(* IEC 61131-3 sources: ia2/library/process-control/pous (part 2) *)

(* ---- fb_pid_3step.st ---- *)
(*
  FB_PID_3STEP — step (3-step) PID: open/close pulse control of a motorized actuator,
  supporting both no-position-feedback (travel-time integral estimate) and
  with-feedback wiring.

  ~ Standard step PID / 3-step output controller (step controller / 3-step PID, driving
  integrating-type actuators such as motorized control valves and motorized dampers),
  found in every major DCS/PLC standard library.

  Purpose: closed-loop control of a motorized actuator (motorized valve / motorized
  damper, which is itself an integrating element: energized it runs open/close, de-energized
  it stops in place). Without a position transmitter, estimate position by integrating
  travel time (pos_fb < 0); with a 4-20 mA position feedback, use it directly.

  Behavior:
    1) Position estimate pos_est: pos_fb >= 0 takes the feedback directly (clamped
       0..100); otherwise integrate from the previous scan's output and the travel time:
       an open pulse adds +100*dt_s/motor_time_s, a close pulse decrements likewise
       (clamped 0..100).
    2) An internal positional PID (reverse-acting e = sp - pv, D on PV with automatic
       3*dt_s PT1 filtering) computes the target position target 0..100; integral
       back-calculation anti-windup; in manual, target tracks pos_est so the return to
       auto is bumpless. For direct-acting scenarios, invert pv/sp externally.
    3) Three-step output: position deviation = target - pos_est;
       > deadband_pct emits an open pulse, < -deadband_pct emits a close pulse, within
       the deadband stop. In auto, once a pulse is emitted it is held at least
       min_pulse_s (to avoid short pulses hammering the contactor); manual jogs
       man_open/man_close pass through (no minimum pulse width, mutually interlocked
       when both are commanded), constrained only by the travel limits. A reversal must
       pass through one scan fully stopped (stop before reversing). At a travel boundary
       (pos_est reaching 0 or 100), stop that direction's pulse immediately.
    Tuning tip: deadband_pct should be larger than the travel corresponding to the
    minimum pulse width (min_pulse_s / motor_time_s * 100%), otherwise it will still
    overshoot and oscillate within the deadband.

  Inputs:
    pv           REAL  process value
    sp           REAL  setpoint
    kp           REAL  proportional gain
    ti_s         REAL  integral time s (0 = no integral)
    td_s         REAL  derivative time s (0 = derivative off)
    dt_s         REAL  sample period s (<= 0 holds this scan, no action)
    motor_time_s REAL  actuator full-travel time s (0->100%; used for estimation and limits)
    min_pulse_s  REAL  minimum pulse width in auto s
    deadband_pct REAL  position deadband % (no action within the deviation deadband)
    auto         BOOL  TRUE auto / FALSE manual jog
    man_open     BOOL  manual open jog (interlocked, no action when commanded with man_close)
    man_close    BOOL  manual close jog
    pos_fb       REAL  position feedback 0..100 % (< 0 = no feedback, use travel estimate)
  Outputs:
    q_open  BOOL  open-direction pulse output
    q_close BOOL  close-direction pulse output
    pos_est REAL  position estimate/feedback 0..100 %
*)
FUNCTION_BLOCK FB_PID_3STEP
  VAR_INPUT
    pv           : REAL;
    sp           : REAL;
    kp           : REAL := 1.0;
    ti_s         : REAL := 0.0;
    td_s         : REAL := 0.0;
    dt_s         : REAL := 0.1;
    motor_time_s : REAL := 60.0;
    min_pulse_s  : REAL := 0.5;
    deadband_pct : REAL := 1.0;
    auto         : BOOL := TRUE;
    man_open     : BOOL := FALSE;
    man_close    : BOOL := FALSE;
    pos_fb       : REAL := -1.0;
  END_VAR
  VAR_OUTPUT
    q_open  : BOOL;
    q_close : BOOL;
    pos_est : REAL;
  END_VAR
  VAR
    i_acc     : REAL; (* positional-PID integral term (back-calculation bumpless) *)
    pv_f      : REAL; (* D-term PT1 filter state *)
    pv_f_prev : REAL;
    t_f       : REAL;
    e         : REAL;
    p_term    : REAL;
    d_term    : REAL;
    target    : REAL; (* PID target position 0..100 *)
    err_pos   : REAL; (* position deviation target - pos_est *)
    pulse_t   : REAL; (* elapsed duration of the current pulse s *)
    open_req  : BOOL; (* open-direction demand this scan *)
    close_req : BOOL;
    init_done : BOOL; (* filter-state first-scan alignment flag *)
  END_VAR

  IF dt_s <= 0.0 THEN
    RETURN; (* invalid sample period: hold *)
  END_IF;

  IF NOT init_done THEN
    pv_f := pv;
    pv_f_prev := pv;
    init_done := TRUE;
  END_IF;

  (* 1) Position estimate: use feedback directly when available; otherwise integrate from the previous scan's output over the travel time *)
  IF pos_fb >= 0.0 THEN
    pos_est := pos_fb;
  ELSE
    IF motor_time_s > 0.0 THEN
      IF q_open THEN
        pos_est := pos_est + 100.0 * dt_s / motor_time_s;
      END_IF;
      IF q_close THEN
        pos_est := pos_est - 100.0 * dt_s / motor_time_s;
      END_IF;
    END_IF;
  END_IF;
  IF pos_est > 100.0 THEN
    pos_est := 100.0;
  ELSIF pos_est < 0.0 THEN
    pos_est := 0.0;
  END_IF;

  (* 2) Positional PID -> target position (reverse-acting; D on PV, automatic 3*dt_s filtering) *)
  t_f := 3.0 * dt_s;
  pv_f := pv_f + dt_s / (t_f + dt_s) * (pv - pv_f);
  e := sp - pv;
  p_term := kp * e;
  d_term := 0.0;
  IF td_s > 0.0 THEN
    d_term := 0.0 - kp * td_s * (pv_f - pv_f_prev) / dt_s;
  END_IF;
  pv_f_prev := pv_f;

  IF auto THEN
    IF ti_s > 0.0 THEN
      i_acc := i_acc + kp * dt_s / ti_s * e;
    END_IF;
    target := p_term + i_acc + d_term;
  ELSE
    target := pos_est; (* Manual: target tracks the current position, bumpless return to auto *)
  END_IF;
  IF target > 100.0 THEN
    target := 100.0;
  ELSIF target < 0.0 THEN
    target := 0.0;
  END_IF;
  IF ti_s > 0.0 OR NOT auto THEN
    i_acc := target - p_term - d_term; (* Back-calculation: anti-windup + bumpless *)
  END_IF;

  (* 3) Three-step output demand *)
  IF auto THEN
    err_pos := target - pos_est;
    open_req := err_pos > deadband_pct;
    close_req := err_pos < 0.0 - deadband_pct;
  ELSE
    open_req := man_open AND NOT man_close; (* Manual jog passes through, interlocked when both commanded *)
    close_req := man_close AND NOT man_open;
  END_IF;

  (* Travel limits: at a boundary, stop emitting that direction's pulse (same in manual/auto) *)
  IF pos_est >= 100.0 THEN
    open_req := FALSE;
  END_IF;
  IF pos_est <= 0.0 THEN
    close_req := FALSE;
  END_IF;

  (* Pulse timing and output: in auto, dropping the demand must satisfy the minimum
     pulse width; in manual, dropping stops immediately; a reversal must pass through
     one scan fully stopped (the current direction drops first, the reverse is allowed
     only on the next scan) *)
  IF q_open OR q_close THEN
    pulse_t := pulse_t + dt_s;
  END_IF;

  IF q_open THEN
    IF pos_est >= 100.0 THEN
      q_open := FALSE; (* at limit, stop *)
    ELSIF NOT open_req AND (NOT auto OR pulse_t >= min_pulse_s) THEN
      q_open := FALSE;
    END_IF;
  ELSIF q_close THEN
    IF pos_est <= 0.0 THEN
      q_close := FALSE;
    ELSIF NOT close_req AND (NOT auto OR pulse_t >= min_pulse_s) THEN
      q_close := FALSE;
    END_IF;
  ELSE
    pulse_t := 0.0;
    IF open_req THEN
      q_open := TRUE;
    ELSIF close_req THEN
      q_close := TRUE;
    END_IF;
  END_IF;
END_FUNCTION_BLOCK

(* ---- fb_pid_pos.st ---- *)
(*
  FB_PID_POS — positional (absolute-output) PID controller with observable p/i/d terms,
  SP weighting, derivative-on-PV (D on PV + PT1 filter), back-calculation anti-windup
  and bumpless transfer.

  ~ Standard positional PID (absolute-output form, observable P/I/D terms, SP weighting
  b, derivative acting on PV), found in every major DCS/PLC standard library.

  Purpose: complements the velocity-form FB_PID -- for loops that need to observe/debug
  the integral term, want SP weighting (b < 1 suppresses the proportional kick on a
  setpoint step), or need an absolute-quantity output downstream. For incremental
  output / cascade relay scenarios, FB_PID is still recommended.

  Algorithm (positional):
    e   := sp - pv (reverse-acting, default); direct = TRUE gives e := pv - sp
    e_p := b*sp - pv (the SP-weighted deviation used only by the P term; reversed when direct)
    p_part := kp * e_p
    i_part := i_part + kp*dt_s/ti_s * e (accumulated when ti_s > 0)
    d_part := -kp*td_s * d(pv_f)/dt (derivative acts on PV: no kick on an SP step;
              pv first passes a PT1 filter, t_dfilt_s <= 0 takes 3*dt_s automatically;
              sign goes positive when direct)
    out := p_part + i_part + d_part + ff, clamped to [out_min, out_max]
  Anti-windup and bumpless (back-calculation): each scan wraps up by back-calculating i_part as
    i_part := out - p_part - d_part - ff
  -- on clamping the integral is pulled back (no windup); in manual/track the output
  follows the supplied value and i_part back-calculates in step, so the return to auto
  has no jump. When ti_s = 0 (no integral), i_part is back-calculated only during
  manual/track (where it is a fixed bias / manual-reset term, not overwritten by
  clamping events during auto, keeping the offset characteristic of P-type control
  stable).
  Mode priority: track > NOT auto (manual) > auto (same as FB_PID).
  Identity: in every mode out = p_part + i_part + d_part + ff (after clamping, except
  on an auto clamping scan with ti_s = 0) -- the sum of the terms is the output,
  intuitive for debugging.

  Inputs:
    pv          REAL  process value
    sp          REAL  setpoint
    kp          REAL  proportional gain
    ti_s        REAL  integral time s (0 = no integral)
    td_s        REAL  derivative time s (0 = derivative off)
    t_dfilt_s   REAL  derivative pre-filter PT1 time constant s (<= 0 = auto 3*dt_s)
    sp_weight_b REAL  SP weighting coefficient b (acts on the P term only; 1 = no weighting,
                      0 = the P term sees pv only -- an SP step gives no proportional kick at all)
    dt_s        REAL  sample period s (<= 0 holds this scan, no action)
    direct      BOOL  TRUE = direct-acting (pv up -> out up), FALSE = reverse-acting
    auto        BOOL  TRUE auto / FALSE manual
    manual_out  REAL  manual output value
    out_min     REAL  output low limit (assumes out_min < out_max)
    out_max     REAL  output high limit
    ff          REAL  feedforward (added to output before clamp)
    track       BOOL  output-tracking enable (highest priority)
    track_value REAL  tracking value
  Outputs:
    out    REAL  control output (clamped in every mode)
    dev    REAL  deviation (reverse-acting sp-pv / direct-acting pv-sp, without SP weighting)
    p_part REAL  proportional term (includes SP weighting)
    i_part REAL  integral term (includes back-calculation correction)
    d_part REAL  derivative term
*)
FUNCTION_BLOCK FB_PID_POS
  VAR_INPUT
    pv          : REAL;
    sp          : REAL;
    kp          : REAL := 1.0;
    ti_s        : REAL := 0.0;
    td_s        : REAL := 0.0;
    t_dfilt_s   : REAL := 0.0;
    sp_weight_b : REAL := 1.0;
    dt_s        : REAL := 0.1;
    direct      : BOOL := FALSE;
    auto        : BOOL := TRUE;
    manual_out  : REAL := 0.0;
    out_min     : REAL := 0.0;
    out_max     : REAL := 100.0;
    ff          : REAL := 0.0;
    track       : BOOL := FALSE;
    track_value : REAL := 0.0;
  END_VAR
  VAR_OUTPUT
    out    : REAL;
    dev    : REAL;
    p_part : REAL;
    i_part : REAL;
    d_part : REAL;
  END_VAR
  VAR
    pv_f      : REAL; (* PV after the D-term PT1 filter *)
    pv_f_prev : REAL; (* previous-scan filtered value, for the backward difference *)
    t_f       : REAL; (* filter time constant actually used *)
    d_pv      : REAL; (* rate of change of the filtered PV, units/s *)
    e         : REAL; (* control deviation (includes the action direction) *)
    e_p       : REAL; (* P-term deviation (SP weighting b) *)
    init_done : BOOL; (* filter-state first-scan alignment flag *)
  END_VAR

  IF dt_s <= 0.0 THEN
    RETURN; (* invalid sample period: hold output and history unchanged *)
  END_IF;

  IF NOT init_done THEN
    pv_f := pv; (* align the filter state: no spurious startup derivative *)
    pv_f_prev := pv;
    init_done := TRUE;
  END_IF;

  (* D-term pre-filter PT1 + backward difference (same core as FB_DERIV) *)
  t_f := t_dfilt_s;
  IF t_f <= 0.0 THEN
    t_f := 3.0 * dt_s;
  END_IF;
  pv_f := pv_f + dt_s / (t_f + dt_s) * (pv - pv_f);
  d_pv := (pv_f - pv_f_prev) / dt_s;
  pv_f_prev := pv_f;

  (* Deviation (by action direction) and the SP-weighted P deviation *)
  IF direct THEN
    e := pv - sp;
    e_p := pv - sp_weight_b * sp;
  ELSE
    e := sp - pv;
    e_p := sp_weight_b * sp - pv;
  END_IF;
  dev := e;

  p_part := kp * e_p;

  d_part := 0.0;
  IF td_s > 0.0 THEN
    (* Derivative acts on PV (no kick on an SP step): reverse-acting, rising pv should push the output down -> negative sign *)
    IF direct THEN
      d_part := kp * td_s * d_pv;
    ELSE
      d_part := 0.0 - kp * td_s * d_pv;
    END_IF;
  END_IF;

  IF track THEN
    (* Output tracking: follows track_value unconditionally, highest priority *)
    out := track_value;
  ELSIF NOT auto THEN
    (* Manual: follows manual_out; the i_part back-calculation guarantees a bumpless return to auto *)
    out := manual_out;
  ELSE
    IF ti_s > 0.0 THEN
      i_part := i_part + kp * dt_s / ti_s * e;
    END_IF;
    out := p_part + i_part + d_part + ff;
  END_IF;

  (* Output clamp *)
  IF out > out_max THEN
    out := out_max;
  ELSIF out < out_min THEN
    out := out_min;
  END_IF;

  (* Back-calculate i_part: makes P+I+D+ff always equal the clamped output -> clamping
     gives anti-windup and manual/track gives bumpless alignment. When ti_s = 0,
     back-calculate only during manual/track (see header note) *)
  IF ti_s > 0.0 OR track OR NOT auto THEN
    i_part := out - p_part - d_part - ff;
  END_IF;
END_FUNCTION_BLOCK

(* ---- fb_pulser.st ---- *)
(*
  FB_PULSER — 周期脉冲发生器。

  用途：料仓空气炮/气锤周期吹扫、周期润滑、心跳输出。
  例：使能后每 period_s 秒输出一个 pulse_len_s 秒宽的脉冲（周期起点先出脉冲）。

  行为：
    enable 时相位 phase_s 以 dt_s 手工累加；phase_s < pulse_len_s 期间 q := TRUE，
    到 period_s 回卷（减法回卷，长期节拍不漂移）。
    NOT enable 或参数非法（period_s/dt_s <= 0）时 q := FALSE 且相位清零
    （重新使能从脉冲开始）。
    pulse_len_s >= period_s 时 q 恒为 TRUE（按定义连续输出）。

  输入：
    enable      BOOL  使能
    period_s    REAL  脉冲周期 s
    pulse_len_s REAL  脉冲宽度 s
    dt_s        REAL  采样周期 s
  输出：
    q BOOL  脉冲输出
*)
FUNCTION_BLOCK FB_PULSER
  VAR_INPUT
    enable      : BOOL;
    period_s    : REAL := 60.0;
    pulse_len_s : REAL := 1.0;
    dt_s        : REAL := 0.1;
  END_VAR
  VAR_OUTPUT
    q : BOOL;
  END_VAR
  VAR
    phase_s : REAL; (* 周期内相位 0..period_s，手工计时替代 TP/TON *)
  END_VAR

  IF NOT enable OR period_s <= 0.0 OR dt_s <= 0.0 THEN
    phase_s := 0.0;
    q := FALSE;
    RETURN;
  END_IF;

  (* 先按当前相位出脉冲（使能首周期立即为 TRUE），再推进相位 *)
  q := phase_s < pulse_len_s;

  phase_s := phase_s + dt_s;
  IF phase_s >= period_s THEN
    phase_s := phase_s - period_s; (* 减法回卷，保持长期节拍 *)
  END_IF;
END_FUNCTION_BLOCK

(* ---- fb_pv_hold.st ---- *)
(*
  FB_PV_HOLD — 坏值保持/替代（bad-PV hold / substitute）。

  ≈ 标准坏值处理块（last-good hold / substitute value，含坏值
  超时降级），测量信号进控制回路前的标准防线，各主流 DCS/PLC
  的输入处理均有同类机制。

  用途：变送器断线/超量程（如 FB_SCALE.fault、FB_MID3.q_fail 取反
  作 good）时给下游回路一个可控的 PV：先保持最后好值渡过抖动，
  超时后按组态保持/替代/跟随，并出 q_bad/q_timeout 供报警与
  回路切手动逻辑使用。

  行为：
    good = TRUE：out := u，记忆最后好值，q_bad/q_timeout 清零，
    坏值计时清零。
    good = FALSE：q_bad := TRUE，坏值计时累加（手工 dt_s）：
      未到 timeout_s：out := 最后好值（短时抖动按保持渡过）；
      到 timeout_s（timeout_s = 0 立即）：q_timeout := TRUE，按 mode：
        mode = 0：继续保持最后好值；
        mode = 1：out := sub_value（替代值，如安全侧设定）；
        mode = 2：out := u（跟随原值——只挂报警牌不干预，
                  下游自行处置）。
    首扫描即坏值时最后好值取当前 u（无更好历史）。
    dt_s <= 0 → 坏值计时不推进（timeout_s > 0 时维持保持段）。

  输入：
    u         REAL  输入（原始 PV）
    good      BOOL  输入有效（FALSE = 坏值；接质量位/断线判定取反）
    mode      REAL  0 = 保持最后好值 / 1 = 替代值 / 2 = 跟随原值
    sub_value REAL  替代值（mode = 1 用）
    timeout_s REAL  坏值持续超时 s（0 = 立即按 mode 动作；> 0 先保持）
    dt_s      REAL  采样周期 s
  输出：
    out       REAL  处理后的 PV
    q_bad     BOOL  坏值中（电平）
    q_timeout BOOL  坏值已超时（mode 已生效）
*)
FUNCTION_BLOCK FB_PV_HOLD
  VAR_INPUT
    u         : REAL;
    good      : BOOL := TRUE;
    mode      : REAL := 0.0;
    sub_value : REAL := 0.0;
    timeout_s : REAL := 0.0;
    dt_s      : REAL := 0.1;
  END_VAR
  VAR_OUTPUT
    out       : REAL;
    q_bad     : BOOL;
    q_timeout : BOOL;
  END_VAR
  VAR
    last_good : REAL; (* 最后好值 *)
    bad_t     : REAL; (* 坏值持续累计时间 s *)
    init_done : BOOL; (* 首扫描播种标志 *)
  END_VAR

  IF NOT init_done THEN
    last_good := u; (* 首扫描即坏值时也以当前 u 作保持值 *)
    init_done := TRUE;
  END_IF;

  IF good THEN
    last_good := u;
    out := u;
    q_bad := FALSE;
    q_timeout := FALSE;
    bad_t := 0.0;
    RETURN;
  END_IF;

  q_bad := TRUE;

  (* 超时前：保持最后好值（短时抖动渡过段） *)
  IF timeout_s > 0.0 THEN
    IF dt_s > 0.0 THEN
      bad_t := bad_t + dt_s;
    END_IF;
    IF bad_t < timeout_s THEN
      out := last_good;
      q_timeout := FALSE;
      RETURN;
    END_IF;
  END_IF;

  (* 超时（或 timeout_s = 0 立即）：按 mode 动作 *)
  q_timeout := TRUE;
  IF mode >= 1.5 THEN
    out := u;         (* 2 = 跟随原值 *)
  ELSIF mode >= 0.5 THEN
    out := sub_value; (* 1 = 替代值 *)
  ELSE
    out := last_good; (* 0 = 保持最后好值 *)
  END_IF;
END_FUNCTION_BLOCK

(* ---- fb_pwm.st ---- *)
(*
  FB_PWM — 时间比例输出（0..100% 指令 → 固定周期占空比通断）。

  ≈ 时间比例输出（time-proportioning / PWM）：连续量 → 周期通断，固态继电器/电磁阀温控惯用。

  用途：PID 输出驱动固态继电器/电磁阀的通断式执行机构：电加热器、
  蒸汽通断阀、加药泵。
  行为：
    相位累加器同 FB_PULSER：phase_s 以 dt_s 累加，到 period_s 减法回卷
    （长期节拍不漂移）；q := phase_s < on_s。
    on_s := u/100 * period_s（u 先钳位 0..100）。
    最小通/断时间（保护接触器/SSR/阀件，按有效占空比钳位实现）：
      0 < on_s < min_on_s            → on_s 提升至 min_on_s；
      0 < period_s - on_s < min_off_s → on_s 压缩至 period_s - min_off_s
      （断侧优先级更高；若 min_on_s + min_off_s > period_s 属参数矛盾，
      实际向断侧让步，极端时恒断——勿如此整定）。
    u <= 0 → 整周期断；u >= 100 → 整周期通（满幅不受最小通断钳位影响）。
    NOT enable 或 period_s/dt_s <= 0 → q := FALSE 且相位清零
    （重新使能从周期起点开始，先通后断）。
    u 变化即时生效（周期内比较门限即变，无需等下个周期）。

  输入：
    u         REAL  指令 0..100 %
    period_s  REAL  PWM 周期 s
    min_on_s  REAL  最小导通时间 s（0 = 不限）
    min_off_s REAL  最小关断时间 s（0 = 不限）
    enable    BOOL  使能
    dt_s      REAL  采样周期 s
  输出：
    q         BOOL  时间比例输出
*)
FUNCTION_BLOCK FB_PWM
  VAR_INPUT
    u         : REAL;
    period_s  : REAL := 10.0;
    min_on_s  : REAL := 0.0;
    min_off_s : REAL := 0.0;
    enable    : BOOL;
    dt_s      : REAL := 0.1;
  END_VAR
  VAR_OUTPUT
    q : BOOL;
  END_VAR
  VAR
    phase_s : REAL; (* 周期内相位，手工计时替代 TP/TON *)
    uc      : REAL;
    on_s    : REAL; (* 本拍有效导通时长 *)
    off_s   : REAL;
  END_VAR

  IF NOT enable OR period_s <= 0.0 OR dt_s <= 0.0 THEN
    phase_s := 0.0;
    q := FALSE;
    RETURN;
  END_IF;

  uc := u;
  IF uc < 0.0 THEN
    uc := 0.0;
  ELSIF uc > 100.0 THEN
    uc := 100.0;
  END_IF;

  on_s := uc * period_s / 100.0;

  (* 最小导通：有效占空比上调（u=0 不受影响） *)
  IF on_s > 0.0 AND on_s < min_on_s THEN
    on_s := min_on_s;
  END_IF;

  (* 最小关断：有效占空比下调（u=100 时 off=0 不触发，保持恒通） *)
  off_s := period_s - on_s;
  IF off_s > 0.0 AND off_s < min_off_s THEN
    on_s := period_s - min_off_s;
    IF on_s < 0.0 THEN
      on_s := 0.0;
    END_IF;
  END_IF;

  q := phase_s < on_s;

  phase_s := phase_s + dt_s;
  IF phase_s >= period_s THEN
    phase_s := phase_s - period_s; (* 减法回卷，保持长期节拍 *)
  END_IF;
END_FUNCTION_BLOCK

(* ---- fb_ramp.st ---- *)
(*
  FB_RAMP — 设定值斜坡发生器（朝固定目标限速逼近）。

  ≈ 标准设定值斜坡发生器（ramp generator）。

  用途：设定值缓变（避免阶跃冲击执行机构/工艺）、升温升压曲线分段执行。
  与 FB_RATE_LIMIT 的区别：本块朝固定 target 走并报告 ramping；
  RATE_LIMIT 连续跟随变化的输入、只钳每秒变化量。

  行为：
    out 以 rate_up（上行）/ rate_dn（下行，传正数）单位/秒逼近 target，
    到达后 ramping := FALSE。速率 = 0 表示该方向直接跳变。
    track 电平有效：out 无条件跟随 track_value 且 ramping := FALSE；
    track 撤销后从当前值续 ramp 到 target（无扰投运惯用：先 track 对中
    当前工艺值，再放开开始斜坡）。
    dt_s <= 0 → 保持。注意 out 初值为 0：投运首拍建议用 track 对中。

  输入：
    target      REAL  目标值
    rate_up     REAL  上行速率 单位/s（0 = 跳变）
    rate_dn     REAL  下行速率 单位/s（传正数；0 = 跳变）
    dt_s        REAL  采样周期 s
    track       BOOL  跟踪使能（电平有效）
    track_value REAL  跟踪值
  输出：
    out     REAL  斜坡输出
    ramping BOOL  斜坡进行中（未到 target）
*)
FUNCTION_BLOCK FB_RAMP
  VAR_INPUT
    target      : REAL;
    rate_up     : REAL := 0.0;
    rate_dn     : REAL := 0.0;
    dt_s        : REAL := 0.1;
    track       : BOOL := FALSE;
    track_value : REAL := 0.0;
  END_VAR
  VAR_OUTPUT
    out     : REAL;
    ramping : BOOL;
  END_VAR
  VAR
    delta : REAL;
    step  : REAL;
  END_VAR

  IF track THEN
    out := track_value; (* 无扰：撤销后从此处续 ramp *)
    ramping := FALSE;
    RETURN;
  END_IF;

  IF dt_s <= 0.0 THEN
    RETURN; (* 保持 *)
  END_IF;

  delta := target - out;
  IF delta > 0.0 THEN
    step := rate_up * dt_s;
    IF rate_up <= 0.0 OR step >= delta THEN
      out := target; (* 速率 0 跳变 / 本拍可达 *)
      ramping := FALSE;
    ELSE
      out := out + step;
      ramping := TRUE;
    END_IF;
  ELSIF delta < 0.0 THEN
    step := rate_dn * dt_s;
    IF rate_dn <= 0.0 OR step >= 0.0 - delta THEN
      out := target;
      ramping := FALSE;
    ELSE
      out := out - step;
      ramping := TRUE;
    END_IF;
  ELSE
    ramping := FALSE;
  END_IF;
END_FUNCTION_BLOCK

(* ---- fb_rampsoak8.st ---- *)
(*
  FB_RAMPSOAK8 — 8 段程序给定发生器（ramp-soak setpoint programmer）。

  ≈ 标准程序给定/曲线给定块（ramp-soak / setpoint programmer，
  升温曲线、热处理曲线、批次温度程序），各主流 DCS/PLC 与程序
  调节仪均有同类块。

  用途：按"斜坡到目标 + 保温"的分段曲线生成设定值，接 FB_PID /
  FB_PID_POS 的 sp 输入：热处理/养护/反应釜升温程序、开停车
  升降负荷曲线。段参数为标量展开 sp1..sp8 / ramp1_s..ramp8_s /
  soak1_s..soak8_s（本方言 FB 作用域数组不能 codegen，见 README
  坑 7；FB_CHAR 同例）。

  行为：
    每段 N：sp 从上一段电平（段 1 从 sp_init）经 rampN_s 线性斜坡到
    spN（rampN_s <= 0 跳变），再保温 soakN_s（soaking = TRUE；
    soakN_s <= 0 即过）。段参数在进段拍锁存——运行中改参数下一段
    生效。
    run 电平有效：TRUE 启动并推进程序；FALSE → 回到初始（seg := 0，
    sp := sp_init，done 清零），再置 TRUE 从段 1 重新开始。
    hold 电平有效：冻结 sp 与段内计时（hold 期间 advance 无效）。
    advance 上升沿：立即跳下一段（从当前 sp 续斜坡，曲线连续）；
    在末段 advance → 完成（或 cyclic 回绕）。
    末段（n_seg 钳 2..8）保温结束：
      cyclic = FALSE → done := TRUE，sp 钉在末段目标，seg := 0，
      保持到 reset 或 run 撤销；
      cyclic = TRUE  → 回绕段 1（从当前 sp 续斜坡，长期循环）。
    reset 电平有效（优先）：回初始同 run 撤销。
    dt_s <= 0 → 段内不推进（启动/advance 沿照常处理）。

  输入：
    sp1..sp8       REAL  各段目标值（标量展开）
    ramp1_s..ramp8_s REAL  各段斜坡时间 s（<= 0 = 跳变）
    soak1_s..soak8_s REAL  各段保温时间 s（<= 0 = 不保温）
    n_seg          REAL  使用段数 2..8（自动钳位）
    run            BOOL  运行（电平；撤销回初始）
    hold           BOOL  暂停（电平；冻结 sp 与计时）
    advance        BOOL  跳段（上升沿）
    reset          BOOL  复位（电平，优先）
    cyclic         BOOL  TRUE = 末段完成后回绕段 1 循环
    sp_init        REAL  起始值（段 1 斜坡的出发电平）
    dt_s           REAL  采样周期 s
  输出：
    sp      REAL  程序设定值输出
    seg     REAL  当前段 1..8（0 = 未运行/已完成）
    soaking BOOL  保温段进行中
    done    BOOL  程序完成（非循环；保持到 reset / run 撤销）
*)
FUNCTION_BLOCK FB_RAMPSOAK8
  VAR_INPUT
    sp1     : REAL := 0.0;
    sp2     : REAL := 0.0;
    sp3     : REAL := 0.0;
    sp4     : REAL := 0.0;
    sp5     : REAL := 0.0;
    sp6     : REAL := 0.0;
    sp7     : REAL := 0.0;
    sp8     : REAL := 0.0;
    ramp1_s : REAL := 0.0;
    ramp2_s : REAL := 0.0;
    ramp3_s : REAL := 0.0;
    ramp4_s : REAL := 0.0;
    ramp5_s : REAL := 0.0;
    ramp6_s : REAL := 0.0;
    ramp7_s : REAL := 0.0;
    ramp8_s : REAL := 0.0;
    soak1_s : REAL := 0.0;
    soak2_s : REAL := 0.0;
    soak3_s : REAL := 0.0;
    soak4_s : REAL := 0.0;
    soak5_s : REAL := 0.0;
    soak6_s : REAL := 0.0;
    soak7_s : REAL := 0.0;
    soak8_s : REAL := 0.0;
    n_seg   : REAL := 2.0;
    run     : BOOL := FALSE;
    hold    : BOOL := FALSE;
    advance : BOOL := FALSE;
    reset   : BOOL := FALSE;
    cyclic  : BOOL := FALSE;
    sp_init : REAL := 0.0;
    dt_s    : REAL := 0.1;
  END_VAR
  VAR_OUTPUT
    sp      : REAL;
    seg     : REAL;
    soaking : BOOL;
    done    : BOOL;
  END_VAR
  VAR
    nn         : REAL; (* 钳位后的段数 2..8 *)
    elapsed_t  : REAL; (* 段内相位计时 s（斜坡/保温各自从 0 起） *)
    level_from : REAL; (* 本段斜坡出发电平 *)
    seg_sp     : REAL; (* 进段锁存的段参数 *)
    seg_ramp_s : REAL;
    seg_soak_s : REAL;
    enter_seg  : REAL; (* 本拍要进入的段号（0 = 不进段） *)
    go_next    : BOOL; (* 本拍段完成/跳段 *)
    adv_edge   : BOOL;
    prev_adv   : BOOL; (* advance 上升沿记忆 *)
  END_VAR

  IF reset THEN
    seg := 0.0;
    soaking := FALSE;
    done := FALSE;
    sp := sp_init;
    elapsed_t := 0.0;
    prev_adv := advance;
    RETURN;
  END_IF;

  adv_edge := advance AND NOT prev_adv;
  prev_adv := advance;

  IF NOT run THEN
    (* 停止：回初始，重新 run 从段 1 开始 *)
    seg := 0.0;
    soaking := FALSE;
    done := FALSE;
    sp := sp_init;
    RETURN;
  END_IF;

  IF done THEN
    RETURN; (* 完成保持：sp 钉在末段目标，等 reset / run 撤销 *)
  END_IF;

  nn := n_seg;
  IF nn < 2.0 THEN
    nn := 2.0;
  ELSIF nn > 8.0 THEN
    nn := 8.0;
  END_IF;

  enter_seg := 0.0;
  go_next := FALSE;

  IF seg < 0.5 THEN
    (* 启动：从 sp_init 进段 1 *)
    sp := sp_init;
    enter_seg := 1.0;
  ELSIF hold THEN
    RETURN; (* 冻结：sp 与计时保持（advance 在 hold 期间无效） *)
  ELSIF adv_edge THEN
    go_next := TRUE; (* 跳段：从当前 sp 续走 *)
  ELSE
    IF dt_s <= 0.0 THEN
      RETURN; (* 采样周期非法：段内不推进 *)
    END_IF;
    elapsed_t := elapsed_t + dt_s;
    IF NOT soaking THEN
      (* 斜坡相位 *)
      IF seg_ramp_s <= 0.0 THEN
        sp := seg_sp; (* 跳变段 *)
        soaking := TRUE;
        elapsed_t := 0.0;
      ELSIF elapsed_t >= seg_ramp_s THEN
        sp := seg_sp;
        soaking := TRUE;
        elapsed_t := elapsed_t - seg_ramp_s; (* 跨相位余量结转 *)
      ELSE
        sp := level_from + (seg_sp - level_from) * elapsed_t / seg_ramp_s;
      END_IF;
    END_IF;
    IF soaking AND elapsed_t >= seg_soak_s THEN
      go_next := TRUE; (* 保温结束 *)
    END_IF;
  END_IF;

  (* 段推进决策：末段 → 完成/回绕；否则进下一段 *)
  IF go_next THEN
    IF seg >= nn - 0.5 THEN
      IF cyclic THEN
        enter_seg := 1.0; (* 回绕：段 1 从当前 sp 续斜坡 *)
      ELSE
        done := TRUE;
        sp := seg_sp; (* 完成：钉在末段目标（提前跳段也直接到位） *)
        seg := 0.0;
        soaking := FALSE;
      END_IF;
    ELSE
      enter_seg := seg + 1.0;
    END_IF;
  END_IF;

  (* 进段：锁存段参数，斜坡从当前 sp 出发 *)
  IF enter_seg > 0.5 THEN
    seg := enter_seg;
    level_from := sp;
    elapsed_t := 0.0;
    soaking := FALSE;
    IF seg <= 1.5 THEN
      seg_sp := sp1;
      seg_ramp_s := ramp1_s;
      seg_soak_s := soak1_s;
    ELSIF seg <= 2.5 THEN
      seg_sp := sp2;
      seg_ramp_s := ramp2_s;
      seg_soak_s := soak2_s;
    ELSIF seg <= 3.5 THEN
      seg_sp := sp3;
      seg_ramp_s := ramp3_s;
      seg_soak_s := soak3_s;
    ELSIF seg <= 4.5 THEN
      seg_sp := sp4;
      seg_ramp_s := ramp4_s;
      seg_soak_s := soak4_s;
    ELSIF seg <= 5.5 THEN
      seg_sp := sp5;
      seg_ramp_s := ramp5_s;
      seg_soak_s := soak5_s;
    ELSIF seg <= 6.5 THEN
      seg_sp := sp6;
      seg_ramp_s := ramp6_s;
      seg_soak_s := soak6_s;
    ELSIF seg <= 7.5 THEN
      seg_sp := sp7;
      seg_ramp_s := ramp7_s;
      seg_soak_s := soak7_s;
    ELSE
      seg_sp := sp8;
      seg_ramp_s := ramp8_s;
      seg_soak_s := soak8_s;
    END_IF;
  END_IF;
END_FUNCTION_BLOCK

(* ---- fb_rate_limit.st ---- *)
(*
  FB_RATE_LIMIT — 变化率限幅器（跟随输入的斜率钳位）。

  ≈ 标准变化率限幅器（velocity/slew limiter）。

  用途：限制连续变化信号的每秒变化量：阀位指令防抖、变频给定缓变、
  前馈量平滑。与 FB_RAMP 的区别：本块跟随持续变化的输入 u（无目标概念），
  只钳 |Δ|/s；RAMP 朝固定 target 走。

  行为：
    delta := u - out 钳位到 ±rate_s*dt_s 后累加：out := out + delta_clamped。
    rate_s <= 0 → 直通；dt_s <= 0 → 保持；
    reset 或首扫描 → out := u（对中，避免投运从 0 全速爬升）。

  输入：
    u      REAL  输入
    rate_s REAL  最大变化率 |单位|/s（0 = 直通）
    dt_s   REAL  采样周期 s
    reset  BOOL  复位/对中（电平有效：out 跟随 u）
  输出：
    out    REAL  限速输出
*)
FUNCTION_BLOCK FB_RATE_LIMIT
  VAR_INPUT
    u      : REAL;
    rate_s : REAL := 0.0;
    dt_s   : REAL := 0.1;
    reset  : BOOL := FALSE;
  END_VAR
  VAR_OUTPUT
    out : REAL;
  END_VAR
  VAR
    delta     : REAL;
    max_step  : REAL;
    init_done : BOOL;
  END_VAR

  IF reset OR NOT init_done THEN
    out := u;
    init_done := TRUE;
    RETURN;
  END_IF;

  IF rate_s <= 0.0 THEN
    out := u; (* 直通 *)
    RETURN;
  END_IF;

  IF dt_s <= 0.0 THEN
    RETURN; (* 保持 *)
  END_IF;

  delta := u - out;
  max_step := rate_s * dt_s;
  IF delta > max_step THEN
    delta := max_step;
  ELSIF delta < 0.0 - max_step THEN
    delta := 0.0 - max_step;
  END_IF;
  out := out + delta;
END_FUNCTION_BLOCK

(* ---- fb_ratio.st ---- *)
(*
  FB_RATIO — 比值站（比值给定器）。

  ≈ 比值站（ratio station）：配比/配料回路惯用块，输出接下游 PID 的 sp。

  用途：配比控制：从动流量设定值 = 主动（wild）流量 × 比值 + 偏置，
  sp 输出接下游 FB_PID 的 sp 输入构成比值回路。
  例：碳化塔石灰乳流量按进气量 0.85 配比跟随。

  公式：sp := clamp(ratio, ratio_min, ratio_max) * wild_flow + bias。
  说明：仅对 ratio 钳位（操作员可调比值的安全限幅），不对 sp 钳位——
  sp 量纲随 wild_flow，下游 PID 自有输出钳位。

  输入：
    wild_flow REAL  主动流量（不受本回路控制的"野"流量）
    ratio     REAL  比值
    ratio_min REAL  比值下限
    ratio_max REAL  比值上限
    bias      REAL  偏置（工程单位）
  输出：
    sp        REAL  从动回路设定值
*)
FUNCTION_BLOCK FB_RATIO
  VAR_INPUT
    wild_flow : REAL;
    ratio     : REAL := 1.0;
    ratio_min : REAL := 0.0;
    ratio_max : REAL := 10.0;
    bias      : REAL := 0.0;
  END_VAR
  VAR_OUTPUT
    sp : REAL;
  END_VAR
  VAR
    ratio_used : REAL;
  END_VAR

  ratio_used := ratio;
  IF ratio_used < ratio_min THEN
    ratio_used := ratio_min;
  ELSIF ratio_used > ratio_max THEN
    ratio_used := ratio_max;
  END_IF;

  sp := ratio_used * wild_flow + bias;
END_FUNCTION_BLOCK

(* ---- fb_runtime.st ---- *)
(*
  FB_RUNTIME — 设备运行小时 + 启动次数统计。

  ≈ 设备运行统计（累计运行小时 + 启动次数），维护保养数据标配。

  用途：泵/风机磨损均衡（hours 接 FB_DUTY2 的 hours_a/b，配 alt_mode=1）、
  维保到期提醒、启停频度统计。
  行为：
    running 为 TRUE 期间 hours := hours + dt_s/3600；
    running 上升沿 starts := starts + 1；
    reset 电平有效，两者清零（优先，复位周期不累计）。
    实例可由调用方放 VAR RETAIN 块下断电保持（同 FB_TOTALIZER 注意事项：
    IA2 retain 按 i32 存取，REAL 小时数的保持精度受此限制；starts 为
    整数计数不受影响）。

  输入：
    running BOOL  设备运行中（接运行反馈，必要时前置 FB_DEBOUNCE）
    reset   BOOL  清零（电平有效，优先；检修换泵后用）
    dt_s    REAL  采样周期 s
  输出：
    hours  REAL  累计运行小时
    starts DINT  累计启动次数
*)
FUNCTION_BLOCK FB_RUNTIME
  VAR_INPUT
    running : BOOL;
    reset   : BOOL := FALSE;
    dt_s    : REAL := 0.1;
  END_VAR
  VAR_OUTPUT
    hours  : REAL;
    starts : DINT;
  END_VAR
  VAR
    prev_run : BOOL; (* 上升沿记忆 *)
  END_VAR

  IF reset THEN
    hours := 0.0;
    starts := 0;
  ELSE
    IF running AND NOT prev_run THEN
      starts := starts + 1;
    END_IF;
    IF running AND dt_s > 0.0 THEN
      hours := hours + dt_s / 3600.0;
    END_IF;
  END_IF;
  prev_run := running;
END_FUNCTION_BLOCK

(* ---- fb_scale.st ---- *)
(*
  FB_SCALE — 线性量程变换：原始计数值 → 工程单位，含 NE43 风格断线提示。

  用途：模拟量输入标定。例如 4-20 mA 采样为原始计数（S7 风格 5530..27648），
  变换为 0..100 % 或 0..5 m 等工程值。

  公式：out := out_min + (raw - raw_min) * (out_max - out_min) / span
        其中 span = MAX(raw_max - raw_min, 1e-6)（内联 IF 实现，防除零）。
  假定 raw_max > raw_min（正向量程）。

  输入：
    raw      REAL  原始计数值（如 AI 通道原值）
    raw_min  REAL  量程下限对应的原始值（4 mA 点）
    raw_max  REAL  量程上限对应的原始值（20 mA 点）
    out_min  REAL  工程量程下限
    out_max  REAL  工程量程上限
    clamp    BOOL  TRUE 时输出钳位在 [out_min, out_max]（支持反向工程量程）
  输出：
    out      REAL  工程值
    fault    BOOL  原始值越界 >5% 量程（NE43 风格断线/超限提示，不锁存）
*)
FUNCTION_BLOCK FB_SCALE
  VAR_INPUT
    raw     : REAL;
    raw_min : REAL := 0.0;
    raw_max : REAL := 27648.0;
    out_min : REAL := 0.0;
    out_max : REAL := 100.0;
    clamp   : BOOL := TRUE;
  END_VAR
  VAR_OUTPUT
    out   : REAL;
    fault : BOOL;
  END_VAR
  VAR
    span   : REAL;
    margin : REAL;
    lo     : REAL;
    hi     : REAL;
  END_VAR

  (* span = MAX(raw_max - raw_min, 1e-6) — 内联 IF 防除零 *)
  span := raw_max - raw_min;
  IF span < 0.000001 THEN
    span := 0.000001;
  END_IF;

  (* NE43 风格越界判定：超出原始量程 5% 以上视为断线/故障 *)
  margin := 0.05 * span;
  fault := (raw < raw_min - margin) OR (raw > raw_max + margin);

  out := out_min + (raw - raw_min) * (out_max - out_min) / span;

  IF clamp THEN
    IF out_min <= out_max THEN
      lo := out_min;
      hi := out_max;
    ELSE
      lo := out_max;
      hi := out_min;
    END_IF;
    IF out < lo THEN
      out := lo;
    ELSIF out > hi THEN
      out := hi;
    END_IF;
  END_IF;
END_FUNCTION_BLOCK

(* ---- fb_select_hl.st ---- *)
(*
  FB_SELECT_HL — 高/低选择器（超驰选择）。

  ≈ 高/低选择器（override selector），超驰控制惯用块。

  用途：超驰（override）控制——两个控制器输出取高/取低共用一个执行机构
  （如压缩机防喘振超驰、压力超驰温度回路）；亦可做双变送器取高/取低。

  行为：select_high = TRUE 取大者，FALSE 取小者；
  a_selected 指示当前输出取自 a（相等时判 a 选中，指示不抖动）。

  输入：
    a           REAL  通道 a（常接主控制器输出）
    b           REAL  通道 b（常接超驰控制器输出）
    select_high BOOL  TRUE = 高选 / FALSE = 低选
  输出：
    out        REAL  选中值
    a_selected BOOL  TRUE = 当前输出取自 a
*)
FUNCTION_BLOCK FB_SELECT_HL
  VAR_INPUT
    a           : REAL;
    b           : REAL;
    select_high : BOOL := TRUE;
  END_VAR
  VAR_OUTPUT
    out        : REAL;
    a_selected : BOOL;
  END_VAR

  IF select_high THEN
    IF a >= b THEN
      out := a;
      a_selected := TRUE;
    ELSE
      out := b;
      a_selected := FALSE;
    END_IF;
  ELSE
    IF a <= b THEN
      out := a;
      a_selected := TRUE;
    ELSE
      out := b;
      a_selected := FALSE;
    END_IF;
  END_IF;
END_FUNCTION_BLOCK

(* ---- fb_split_range.st ---- *)
(*
  FB_SPLIT_RANGE — 分程输出：一个调节器输出按 split 点分配到两个阀。

  ≈ 分程输出（split range）：一个调节输出按区段驱动两个阀（加热/冷却、大小阀）。

  用途：一个 PID 驱动两个执行机构：大小阀扩量程（顺序分程，
  reverse_b := FALSE），或加热/冷却、进料/回流互补型分程
  （reverse_b := TRUE，按执行机构气开气关与 PID 作用方向整定）。

  行为（u 先钳位 0..100，两输出亦钳位 0..100）：
    out_a：u 在 [0, split] 内 0→100 线性，u >= split 后保持 100。
    out_b：u 在 [split, 100] 内 0→100 线性，u <= split 时为 0；
           reverse_b = TRUE 时 B 段反转为 100→0（含段外端值保持，
           即 u <= split 时 out_b = 100，输出连续无跳变）。
    曲线示意（split = 50）：
      reverse_b = FALSE（大小阀顺序分程）：
        u:     0 …… 50 …… 100
        out_a: 0 → 100 ┤ 保持 100
        out_b: 0   0   ├ 0 → 100
      reverse_b = TRUE（互补型，B 先全开后渐关）：
        u:     0 …… 50 …… 100
        out_a: 0 → 100 ┤ 保持 100
        out_b: 100 100 ├ 100 → 0
    退化：split <= 0 → A 段无量程（u > 0 即 100）；split >= 100 → B 段
    无量程（u >= 100 才动作）。split 应整定在 (0, 100) 内。

  输入：
    u         REAL  调节器输出 0..100
    split     REAL  分程点 %（B 阀起点）
    reverse_b BOOL  TRUE = B 阀在其分程段内反作用（100→0）
  输出：
    out_a     REAL  A 阀开度 0..100
    out_b     REAL  B 阀开度 0..100
*)
FUNCTION_BLOCK FB_SPLIT_RANGE
  VAR_INPUT
    u         : REAL;
    split     : REAL := 50.0;
    reverse_b : BOOL := TRUE;
  END_VAR
  VAR_OUTPUT
    out_a : REAL;
    out_b : REAL;
  END_VAR
  VAR
    uc     : REAL; (* 钳位后的输入 *)
    span_b : REAL;
  END_VAR

  (* 输入钳位 0..100 *)
  uc := u;
  IF uc < 0.0 THEN
    uc := 0.0;
  ELSIF uc > 100.0 THEN
    uc := 100.0;
  END_IF;

  (* A 阀：[0, split] 内 0→100 *)
  IF split > 0.0 THEN
    out_a := uc * 100.0 / split;
  ELSE
    (* 退化：A 无分程段 *)
    IF uc > 0.0 THEN
      out_a := 100.0;
    ELSE
      out_a := 0.0;
    END_IF;
  END_IF;
  IF out_a < 0.0 THEN
    out_a := 0.0;
  ELSIF out_a > 100.0 THEN
    out_a := 100.0;
  END_IF;

  (* B 阀：[split, 100] 内 0→100 *)
  span_b := 100.0 - split;
  IF span_b > 0.0 THEN
    out_b := (uc - split) * 100.0 / span_b;
  ELSE
    (* 退化：B 无分程段 *)
    IF uc >= split THEN
      out_b := 100.0;
    ELSE
      out_b := 0.0;
    END_IF;
  END_IF;
  IF out_b < 0.0 THEN
    out_b := 0.0;
  ELSIF out_b > 100.0 THEN
    out_b := 100.0;
  END_IF;

  (* B 段反作用（钳位后再反转，段外保持端值，输出连续） *)
  IF reverse_b THEN
    out_b := 100.0 - out_b;
  END_IF;
END_FUNCTION_BLOCK

(* ---- fb_sqrt_flow.st ---- *)
(*
  FB_SQRT_FLOW — 差压流量开方提取。

  ≈ 差压流量开方提取（square-root extraction）+ 小流量切除，DCS 模拟量处理惯用块。

  用途：孔板/文丘里/喷嘴等差压式流量测量：流量与差压的平方根成正比。
  公式：flow := flow_max * SQRT(dp_pct / 100.0)；dp_pct <= cutoff_pct → flow := 0。
  说明：
    cutoff_pct 为小流量切除：低差压区开方增益趋于无穷，噪声放大严重，
    惯例直接切零。默认 6.25%（差压）↔ 25%（流量）切除点。
    dp_pct <= 0 按 0 处理；dp_pct > 100 不截断（允许量程外开方延伸，
    需要硬限时调用方自行钳位）。
    SQRT() 为本方言内建函数（已经 cs project check 含 codegen 验证可用）。

  输入：
    dp_pct     REAL  差压 %（0..100，常接 FB_SCALE 输出）
    flow_max   REAL  100% 差压对应的流量工程值
    cutoff_pct REAL  小流量切除阈值 %（差压百分数）
  输出：
    flow       REAL  流量工程值
*)
FUNCTION_BLOCK FB_SQRT_FLOW
  VAR_INPUT
    dp_pct     : REAL;
    flow_max   : REAL := 100.0;
    cutoff_pct : REAL := 6.25;
  END_VAR
  VAR_OUTPUT
    flow : REAL;
  END_VAR

  IF dp_pct <= cutoff_pct OR dp_pct <= 0.0 THEN
    flow := 0.0; (* 小流量切除 *)
    RETURN;
  END_IF;

  flow := flow_max * SQRT(dp_pct / 100.0);
END_FUNCTION_BLOCK

(* ---- fb_stats.st ---- *)
(*
  FB_STATS — running statistics: min/max/mean/standard deviation (Welford single-pass recurrence).

  ~ Standard statistics block (min/max/average/standard deviation), found in every
  major platform's standard library; this block uses Welford's single-pass
  recurrence -- no arrays, numerically stable.

  Purpose: quality-data statistics (batch temperature mean/spread), measurement
  noise-level assessment, commissioning-time signal profiling (feed FB_AVG_TIME for
  the time average, feed this block for the full-run distribution).
  Behavior (counted by "sample", not consuming dt_s: each scan with enable TRUE counts as 1 sample):
    Welford recurrence (scalar, single-pass, avoiding the precision disaster of
    subtracting squares of large numbers):
      n := n + 1; delta := u - avg; avg := avg + delta / n;
      m2 := m2 + delta * (u - avg)
    sd := SQRT(m2 / n) -- population standard deviation (divide by n, not n-1):
    process monitoring cares about the spread magnitude, the two are indistinguishable
    at large sample counts, and dividing by n is the most direct form in a single-pass
    recurrence.
    reset level-active: clears and re-seeds on the next enabled sample (vmin/vmax/avg
    take that sample's value).
    Note: n is a REAL count; in single precision, after about 1.6E7 samples (about 19
    days at a 100 ms sample) the +1 stops taking effect and the statistics freeze --
    for long-term running, reset per shift / per day.

  Inputs:
    u      REAL  input sample
    enable BOOL  sampling enable (a FALSE scan counts no sample, outputs hold)
    reset  BOOL  clear (level-active, takes priority; re-seeds on the next enabled sample)
  Outputs:
    vmin REAL  minimum value
    vmax REAL  maximum value
    avg  REAL  arithmetic mean
    sd   REAL  population standard deviation
    n    REAL  samples counted so far
*)
FUNCTION_BLOCK FB_STATS
  VAR_INPUT
    u      : REAL;
    enable : BOOL := TRUE;
    reset  : BOOL := FALSE;
  END_VAR
  VAR_OUTPUT
    vmin : REAL;
    vmax : REAL;
    avg  : REAL;
    sd   : REAL;
    n    : REAL;
  END_VAR
  VAR
    m2     : REAL; (* Welford second-order accumulator sum of (u-avg)*(u-avg') *)
    delta  : REAL;
    delta2 : REAL;
  END_VAR

  IF reset THEN
    n := 0.0;
    avg := 0.0;
    m2 := 0.0;
    sd := 0.0;
    vmin := 0.0;
    vmax := 0.0;
    RETURN;
  END_IF;

  IF NOT enable THEN
    RETURN; (* counts no sample: outputs hold *)
  END_IF;

  IF n <= 0.0 THEN
    (* Seed on the first sample *)
    n := 1.0;
    avg := u;
    m2 := 0.0;
    sd := 0.0;
    vmin := u;
    vmax := u;
    RETURN;
  END_IF;

  n := n + 1.0;
  delta := u - avg;
  avg := avg + delta / n;
  delta2 := u - avg;
  m2 := m2 + delta * delta2;
  sd := SQRT(m2 / n);

  IF u < vmin THEN
    vmin := u;
  END_IF;
  IF u > vmax THEN
    vmax := u;
  END_IF;
END_FUNCTION_BLOCK

(* ---- fb_totalizer.st ---- *)
(*
  FB_TOTALIZER — 流量累积器：m3/h 瞬时流量 → m3 累积量。

  用途：进水/进料流量累计、班产/批量计量。
  实例可由调用方放在 VAR RETAIN 块下，使 total 随实例一起断电保持
  （IA2 将 RETAIN 变量快照到 state/retain.json）。

  公式：total := total + flow * dt_s / 3600.0（reset 优先，复位周期不累加）。
  说明：flow 为负时照常累加（允许双向计量）；dt_s <= 0 时不累加。

  输入：
    flow  REAL  瞬时流量 m3/h
    dt_s  REAL  采样周期 s
    reset BOOL  累积清零（电平有效，优先于累加）
  输出：
    total REAL  累积量 m3
*)
FUNCTION_BLOCK FB_TOTALIZER
  VAR_INPUT
    flow  : REAL;
    dt_s  : REAL := 0.1;
    reset : BOOL;
  END_VAR
  VAR_OUTPUT
    total : REAL;
  END_VAR

  IF reset THEN
    total := 0.0;
  ELSIF dt_s > 0.0 THEN
    total := total + flow * dt_s / 3600.0;
  END_IF;
END_FUNCTION_BLOCK

(* ---- fb_valve.st ---- *)
(*
  FB_VALVE — 开关阀（两位阀）控制，带行程超时与双限位故障监视。

  用途：气动/电动开关阀的标准封装，ZSO/ZSC 双限位回讯。
  例：进料阀开到位才允许下游启动；行程超时报阀卡。

  行为：
    1) 故障监视：
       - zso 与 zsc 同时为 TRUE → 限位开关故障，立即 fault；
       - 命令位置与限位回讯不一致（开阀未见 zso / 关阀未见 zsc）持续
         travel_timeout_s（手工 dt_s 累加计时）→ 行程超时 fault；
       - 外部故障 fault_in → fault。均锁存，reset 且 fault_in 消除后清除。
    2) 命令锁存：cmd_open 在 remote 且无故障时置位 out_open；
       cmd_close 或 fault 复位（故障时故障安全关阀，关阀优先）。
    3) 状态字 status：0 关到位 / 1 行程中 / 2 开到位 / 3 故障。

  输入：
    cmd_open         BOOL  开阀命令
    cmd_close        BOOL  关阀命令（优先）
    remote           BOOL  远程允许（仅闸开阀）
    zso              BOOL  开到位限位（Zero Switch Open）
    zsc              BOOL  关到位限位（Zero Switch Closed）
    fault_in         BOOL  外部故障输入
    reset            BOOL  故障复位
    travel_timeout_s REAL  行程超时 s
    dt_s             REAL  采样周期 s
  输出：
    out_open BOOL  开阀输出（TRUE 开 / FALSE 关）
    fault    BOOL  故障（锁存）
    status   INT   0 关到位 / 1 行程中 / 2 开到位 / 3 故障
*)
FUNCTION_BLOCK FB_VALVE
  VAR_INPUT
    cmd_open         : BOOL;
    cmd_close        : BOOL;
    remote           : BOOL := TRUE;
    zso              : BOOL;
    zsc              : BOOL;
    fault_in         : BOOL;
    reset            : BOOL;
    travel_timeout_s : REAL := 30.0;
    dt_s             : REAL := 0.1;
  END_VAR
  VAR_OUTPUT
    out_open : BOOL;
    fault    : BOOL;
    status   : INT;
  END_VAR
  VAR
    travel_t : REAL; (* 未到位累计时间 s *)
    in_pos   : BOOL;
  END_VAR

  (* 1) 故障监视 *)
  IF zso AND zsc THEN
    fault := TRUE; (* 双限位同时有效：限位开关故障 *)
  END_IF;

  in_pos := (out_open AND zso) OR (NOT out_open AND zsc);
  IF in_pos THEN
    travel_t := 0.0;
  ELSE
    travel_t := travel_t + dt_s;
  END_IF;
  IF travel_timeout_s > 0.0 AND travel_t >= travel_timeout_s THEN
    fault := TRUE; (* 行程超时：阀卡/限位丢失 *)
  END_IF;

  IF fault_in THEN
    fault := TRUE;
  END_IF;
  IF reset AND NOT fault_in THEN
    fault    := FALSE;
    travel_t := 0.0;
  END_IF;

  (* 2) 命令锁存（关阀/故障优先，故障安全关阀） *)
  IF cmd_open AND remote AND NOT fault THEN
    out_open := TRUE;
  END_IF;
  IF cmd_close OR fault THEN
    out_open := FALSE;
  END_IF;

  (* 3) 状态字 *)
  IF fault THEN
    status := 3;
  ELSIF out_open AND zso THEN
    status := 2;
  ELSIF NOT out_open AND zsc THEN
    status := 0;
  ELSE
    status := 1;
  END_IF;
END_FUNCTION_BLOCK
